FUNCTION_BLOCK MockSerializableArray IMPLEMENTS I_Serializable
VAR
	_name : STRING;
	_age : INT;
END_VAR

PROPERTY PUBLIC Age : INT
GET
Age := _age;
END_GET
SET
_age := Age;
END_SET
END_PROPERTY

METHOD FB_init : BOOL
VAR_INPUT
	bInitRetains : BOOL; // if TRUE, the retain variables are initialized (warm start / cold start)
	bInCopyCode : BOOL;  // if TRUE, the instance afterwards gets moved into the copy code (online change)
	Name : STRING;
	Age : INT;
END_VAR
_name := Name;
_age := Age;
END_METHOD

PROPERTY PUBLIC Name : STRING
GET
Name := _name;
END_GET
SET
_name := Name;
END_SET
END_PROPERTY

METHOD SerializeWith
VAR_INPUT
	Serializer : I_Serializer;
END_VAR
Serializer.StartArray().AddString(_name).AddInt(_age).EndArray();
END_METHOD

END_FUNCTION_BLOCK

(* stored: Version 1.1.0.1, ProductVersion 3.1.4024.12
   POU MockSerializableArray: Id {dcea679a-a882-4d11-b8d5-fb38495441cf}, SpecialFunc None
   Folder Constructor: Id {feed1b06-6326-4091-a8f3-72bcb1faf80d}
   Property Age: Id {4b8e55b4-c4ce-48b3-b170-34d025712fe1}
   Get Get: Id {b7af2ea5-4b1a-4b84-876e-d5ac4a07746d}
   Set Set: Id {11199343-8167-4825-8ca1-33d93a1007f8}
   Method FB_init: Id {64a2327f-6556-45c3-a5e3-ace48a689b07}
   Property Name: Id {30162b29-73b9-484c-8e39-b6c853eabe3d}
   Get Get: Id {4c50f123-b70b-40b8-8394-fdefc251823f}
   Set Set: Id {0e68035a-9938-427a-a276-0d7d13b8b8e5}
   Method SerializeWith: Id {242fc345-6536-4eeb-b81b-3e6149ab41da} *)
